// TIA Portal project "Set-Reset ile 2 Yönlü Motor Uygulaması" (V18)

(* hardware
DEVICE "S7-1200 station_1"  S7-1200 Station
   slot 0: "Rack_0"  S7-1200 Rack  Rack  V1.0
   slot 1: "PLC_1"  CPU 1214C AC/DC/Rly  6ES7 214-1BG40-0XB0  V4.6
*)

// ===== PLC "PLC_1"  CPU 1214C AC/DC/Rly =====

VAR_GLOBAL   // PLC tag table "Default tag table"
   "Stop" AT %I0.0 : Bool;
   "Start_1" AT %I0.1 : Bool;
   "Start_2" AT %I0.2 : Bool;
   "Motor_1" AT %Q0.0 : Bool;
   "Start_3" AT %I0.3 : Bool;
   "Saat Yönünde" AT %Q0.1 : Bool;
   "Saatin Tersi Yönde" AT %Q0.2 : Bool;
   "Aşırı Akım Koruma" AT %I0.7 : Bool;
   "Motor_4" AT %Q0.3 : Bool;
   "Start_4" AT %I0.4 : Bool;
END_VAR

ORGANIZATION_BLOCK "Main"   // OB1, LAD, ProgramCycle
TITLE = "Main Program Sweep (Cycle)"
{ S7_Optimized_Access := 'TRUE' }
VERSION : 0.1
// Motor iki start butonu ile iki ayrı yönde çalıştırılacaktır. 
// Her buton bir yönde çalışma içindir. 
// Emniyet olarak kontak emniyeti kullanılacaktır. 
// Stop butonu ile motorun durması sağlanacaktır. 
// Set – Reset komutları kullanılarak devre tasarlanacaktır.
   VAR_INPUT
      Initial_Call : Bool;   // Initial call of this OB
      Remanence : Bool;   // =True, if remanent data are available
   END_VAR
BEGIN

REGION Network 1
   // Saat yönünde dönecek ama saatin tersi yönde dönerken çalışmayacak.
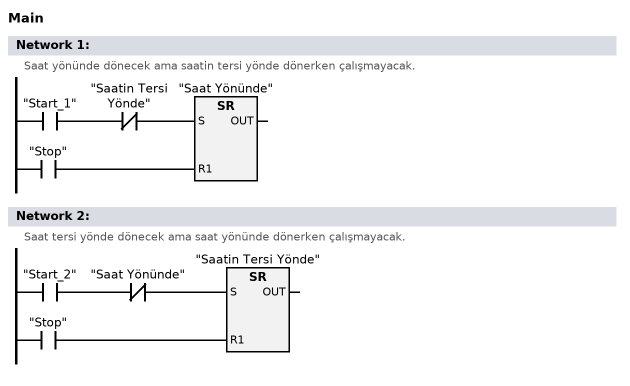
   RUNG wire#powerrail
      Contact( "Start_1" )
      I_Contact( "Saatin Tersi Yönde" )
      S_SR(operand := "Saat Yönünde", r1 := wire#w1)
   END_RUNG
   RUNG wire#powerrail
      Contact( "Stop" )
   END_RUNG wire#w1
   // the same network as SCL:
   IF "Start_1" AND NOT "Saatin Tersi Yönde" THEN
       "Saat Yönünde" := TRUE;   // SR flip-flop
   END_IF;
   IF "Stop" THEN "Saat Yönünde" := FALSE; END_IF;
END_REGION

REGION Network 2
   // Saat tersi yönde dönecek ama saat yönünde dönerken çalışmayacak.
   RUNG wire#powerrail
      Contact( "Start_2" )
      I_Contact( "Saat Yönünde" )
      S_SR(operand := "Saatin Tersi Yönde", r1 := wire#w1)
   END_RUNG
   RUNG wire#powerrail
      Contact( "Stop" )
   END_RUNG wire#w1
   // the same network as SCL:
   IF "Start_2" AND NOT "Saat Yönünde" THEN
       "Saatin Tersi Yönde" := TRUE;   // SR flip-flop
   END_IF;
   IF "Stop" THEN "Saatin Tersi Yönde" := FALSE; END_IF;
END_REGION
END_ORGANIZATION_BLOCK